TYPE ST_scope_info :
STRUCT
	is_connected:BOOL;
	is_ready:BOOL;
	id:UINT;
	scope_deg:UINT;
	scope_up_down:UINT;
	scope_gravity_angle:INT;
	scope_name:STRING;
END_STRUCT
END_TYPE

(* stored: Version 1.1.0.1, ProductVersion 3.1.4024.11
   DUT ST_scope_info: Id {60a07ad3-869b-4fdd-acd6-46198f3ed385} *)
